(* IEC 61131-3 sources: BODAS-HelloWorld/extracted_st/bodas_rc18_12_40/plc_logic/application/02_easyconfig/easyconfig_import/bds_sysio_ec/bds_sysio_ec_gvl, 1 file *)

(* ---- bds_sysIo_ec_gvl.st ---- *)
(* --- Interface --- *)
{attribute 'qualified_only' := ''}
VAR_GLOBAL CONSTANT
    BDS_SYSIO_FI_SHUNT_NUM_SIGNALS_D : UINT := bds_sys_do_signal_te.SHUNT1_EN;
END_VAR
